(* Schneider Machine Expert - Basic project Toggle SW LED, file version 1.8.0.0 *)

HARDWARE
  Cpu 0: TM221CE16R
  EthernetConfiguration: NetworkName=M221, IpAllocationMode=FixedAddress, IpAddress=0.0.0.0, SubnetMask=0.0.0.0
  SerialLineConfiguration: Baud=Baud19200, Parity=ParityEven, DataBits=DataBits8, StopBits=StopBits1, PhysicalMedium=PhysicalMediumRs485, TransmissionMode=TransmissionModeModbusRtu, SlaveId=1, Addressing=SlaveAddressing
  MastTask: UsePeriodScanMode=false, PeriodScan=100
  FastTask: Period=255
  CpuBehavior: StartingMode=StartAsPreviousState, AutoSaveRamOnEeprom=true, WatchdogPeriod=250

SYMBOLS  (address, symbol, comment, settings)
  %I0.0     SW_GREEN

POU New POU
  (* SectionNumber=1 *)

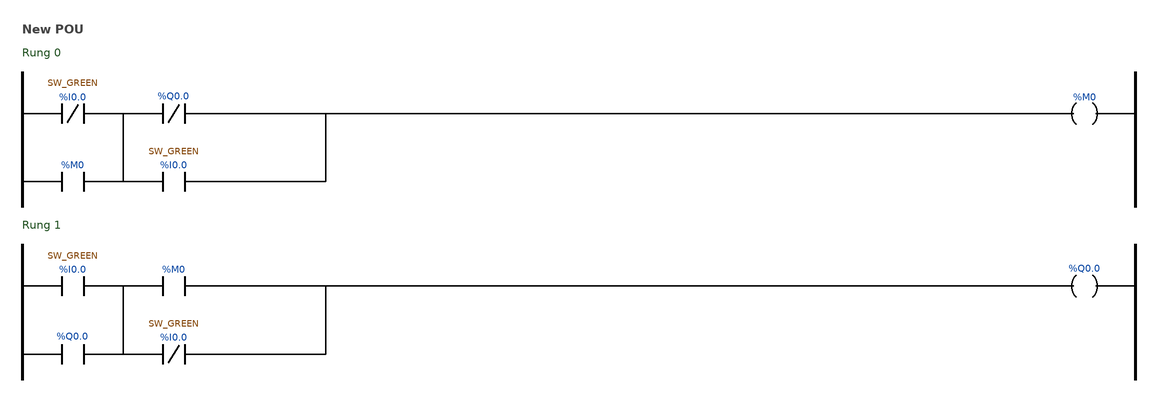

// Rung 0
  LDN %I0.0               (* SW_GREEN *)
  OR %M0
  AND(N %Q0.0
  OR %I0.0                (* SW_GREEN *)
  )
  ST %M0
  // as ST:
  //   %M0 := (NOT SW_GREEN OR %M0) AND (NOT %Q0.0 OR SW_GREEN);

// Rung 1
  LD %I0.0                (* SW_GREEN *)
  OR %Q0.0
  AND( %M0
  ORN %I0.0               (* SW_GREEN *)
  )
  ST %Q0.0
  // as ST:
  //   %Q0.0 := (SW_GREEN OR %Q0.0) AND (%M0 OR NOT SW_GREEN);
